(* CoDeSys 2.3.9.41 project: warm.pro *)
(* Libraries: STANDARD.LIB 4.10.05 10:14:46, IECSFC.LIB 13.4.06 14:51:28, SYSLIBTIME.LIB 20.2.06 13:31:16, SYSTASKINFO.LIB 20.2.06 13:31:38, ANALYZATION.LIB 5.10.99 08:05:06, SYSLIBCALLBACK.LIB 20.2.06 13:31:08 *)

(* PLC configuration (modules and I/O channels)
AT %IX0.0 [BitInput]
AT %IX0.1 [BitInput]
AT %IX0.2 [BitInput]
AT %IX0.3 [BitInput]
AT %IX0.4 [BitInput]
AT %IX0.5 [BitInput]
DO0_nurtureValve AT %QX1.0 [BitOutput]
DO1_genatsuValve AT %QX1.1 [BitOutput]
AT %QX1.2 [BitOutput]
AT %QX1.3 [BitOutput]
Special output [ID104] node 2, in %IB2 out %QB2 {Visibility = No; PinCount = 1}
  AT %QX2.0 [BitOutput] Special output
AI0_presIN AT %ID3.0 [FloatInput] Value
AT %IW3.1 [WordInput] Circular time
Analog Input [ID107] node 0, in %IB3.0 out %QB3.0
AI1_presOUT AT %ID4.0 [FloatInput] Value
AT %IW4.1 [WordInput] Circular time
Analog Input [ID107] node 0, in %IB4.0 out %QB4.0
AI2_outsideTemp AT %ID5.0 [FloatInput] Value
AT %IW5.1 [WordInput] Circular time
Analog Input [ID107] node 0, in %IB5.0 out %QB5.0
AT %ID6.0 [FloatInput] Value
AT %IW6.1 [WordInput] Circular time
Analog Input [ID107] node 0, in %IB6.0 out %QB6.0
Analog output [ID106] node 7, in %IB7 out %QB7 {DAC_Type = Voltage 0-10 B; Analog_offset_correction = 0; Analog_full_range_correction = 0; SafeValueFloat = 0; Visibility = No}
  AT %QD7.0 [FloatOutput] Value
Analog output [ID106] node 8, in %IB8 out %QB8 {DAC_Type = Voltage 0-10 B; Analog_offset_correction = 0; Analog_full_range_correction = 0; SafeValueFloat = 0; Visibility = No}
  AT %QD8.0 [FloatOutput] Value
ModBus (Master) [MODBUS_MASTER_ID450] node 9, in %IB9 out %QB9 {Visibility = No}
  AT %QD9.0 [DWordOutput] Last address
  AT %QW9.1 [WordOutput] Last error
  RS-485-1 [COM1_USART] node 0, in %IB9.0 out %QB9.0 {CommunicationSpeed = 11520; Parity = NO PARITY CHECK; BitLength = 8 bits; StopLength = Two stop bits; InterfaceType = RS485; FrameOriented = RTU; Timeout = 0; Visibility = No}
  Universal Modbus device [ID2000] node 1, in %IB9.1 out %QB9.1 {ModuleIP = 10:0:0:223; ServiceTimeout = 150; TCPport = 502; NetMode = Serial; ModuleSlaveAddress = 3; RequestType = By poll time; PeriodOfService = 3000; Visibility = No; RepeatCounter = 0; ByteSequence = Native}
    AT %QB9.1.0 [ComChannel] Command (0xff - Start)
trm1_temperature AT %IW9.1.0.0 [WordInput]
trm1_setpoint AT %IW9.1.1.0 [WordInput]
trm1_state AT %IW9.1.2.0 [WordInput]
trm1_writeSetpoint AT %QW9.1.3.0 [WordOutput]
Universal Modbus device [ID2000] node 2, in %IB9.2 out %QB9.2 {ModuleIP = 10:0:0:223; ServiceTimeout = 150; TCPport = 502; NetMode = Serial; ModuleSlaveAddress = 4; RequestType = By poll time; PeriodOfService = 3000; Visibility = No; RepeatCounter = 0; ByteSequence = Native}
  AT %QB9.2.0 [ComChannel] Command (0xff - Start)
trm2_temperature AT %IW9.2.0.0 [WordInput]
trm2_setpoint AT %IW9.2.1.0 [WordInput]
trm2_state AT %IW9.2.2.0 [WordInput]
trm2_writeSetpoint AT %QW9.2.3.0 [WordOutput]
Universal Modbus device [ID2000] node 3, in %IB9.3 out %QB9.3 {ModuleIP = 10:0:0:223; ServiceTimeout = 150; TCPport = 502; NetMode = Serial; ModuleSlaveAddress = 5; RequestType = By poll time; PeriodOfService = 2000; Visibility = No; RepeatCounter = 0; ByteSequence = Trace_mode}
  AT %QB9.3.0 [ComChannel] Command (0xff - Start)
fc_frequency AT %IW9.3.0.0 [WordInput]
fc_setpoint AT %ID9.3.1.0 [DWordInput]
fc_power AT %ID9.3.2.0 [DWordInput]
fc_currency AT %ID9.3.3.0 [DWordInput]
fc_pressure AT %ID9.3.4.0 [DWordInput]
fc_writeSetpoint AT %QD9.3.5.0 [DWordOutput]
Debug RS-232 [DEBUG_USART] node 0, in %IB10.0.0 out %QB10.0.0 {CommunicationSpeed = 11520; Parity = EVEN; BitLength = 8 bits; StopLength = One stop bit; InterfaceType = RS232; FrameOriented = RTU; Timeout = 0; Visibility = No}
AT %QB10.1.0 [ByteOutput]
AT %QB10.2.0 [ByteOutput]
AT %QB10.3.0 [ByteOutput]
AT %QB10.4.0 [ByteOutput]
pan_weekDays AT %QB10.5.0 [ByteOutput]
pan_holyDays AT %QB10.6.0 [ByteOutput]
2 byte [Register] node 7, in %IB10.7 out %QB10.7
  pan_trm1_temp AT %QW10.7.0 [WordOutput]
  pan_trm1_set AT %QW10.8.0 [WordOutput]
  pan_trm2_temp AT %QW10.9.0 [WordOutput]
  pan_trm2_set AT %QW10.10.0 [WordOutput]
  pan_fc_freq AT %QW10.11.0 [WordOutput]
  pan_fc_curr AT %QW10.12.0 [WordOutput]
  pan_fc_pow AT %QW10.13.0 [WordOutput]
  pan_fc_pres AT %QW10.14.0 [WordOutput]
  pan_fc_set AT %QW10.15.0 [WordOutput]
  pan_presIN_4ma AT %QW10.16.0 [WordOutput]
  pan_presIN_20ma AT %QW10.17.0 [WordOutput]
  pan_presOUT_4ma AT %QW10.18.0 [WordOutput]
  pan_presOUT_20ma AT %QW10.19.0 [WordOutput]
  pan_weekday_set AT %QW10.20.0 [WordOutput]
  pan_holyday_set AT %QW10.21.0 [WordOutput]
  pan_weekday_onHH AT %QW10.22.0 [WordOutput]
  pan_weekday_onMM AT %QW10.23.0 [WordOutput]
  pan_holyday_onHH AT %QW10.24.0 [WordOutput]
  pan_holyday_onMM AT %QW10.25.0 [WordOutput]
  pan_weekday_offHH AT %QW10.26.0 [WordOutput]
  pan_weekday_offMM AT %QW10.27.0 [WordOutput]
  pan_holyday_offHH AT %QW10.28.0 [WordOutput]
  pan_holyday_offMM AT %QW10.29.0 [WordOutput]
  pan_soldierTime AT %QW10.30.0 [WordOutput]
  pan_airLow AT %QW10.31.0 [WordOutput]
  pan_trmLow AT %QW10.32.0 [WordOutput]
  pan_airHigh AT %QW10.33.0 [WordOutput]
  pan_trmHigh AT %QW10.34.0 [WordOutput]
  pan_nurtureHigh AT %QW10.35.0 [WordOutput]
  pan_nurtureLow AT %QW10.36.0 [WordOutput]
  pan_genatsuHigh AT %QW10.37.0 [WordOutput]
  pan_genatsuLow AT %QW10.38.0 [WordOutput]
  pan_presIN AT %QW10.39.0 [WordOutput]
  pan_presOUT AT %QW10.40.0 [WordOutput]
  pan_outsideTemp AT %QW10.41.0 [WordOutput]
  pan_tempShift AT %QW10.42.0 [WordOutput]
  pan_currHH AT %QW10.43.0 [WordOutput]
  pan_currMIN AT %QW10.44.0 [WordOutput]
  pan_currSS AT %QW10.45.0 [WordOutput]
  pan_currDD AT %QW10.46.0 [WordOutput]
  pan_currMM AT %QW10.47.0 [WordOutput]
  pan_currYY AT %QW10.48.0 [WordOutput]
  pan_setHH AT %QW10.49.0 [WordOutput]
  pan_setMIN AT %QW10.50.0 [WordOutput]
  pan_setSS AT %QW10.51.0 [WordOutput]
  pan_setDD AT %QW10.52.0 [WordOutput]
  pan_setMM AT %QW10.53.0 [WordOutput]
  pan_setYY AT %QW10.54.0 [WordOutput]
  pan_genatsuOmakeHigh AT %QW10.55.0 [WordOutput]
  ID4002 byte8IB
8%QB
8%MB
8%Mpan_genatsuOmakeLow AT %QW10.56.0 [WordOutput]
*)

(* Global variable list: Global_Variables *)
VAR_GLOBAL
(* Times *)
	GetTime: CurTimeEx;
	TimeAndDate: SystemTimeDate;
	Sys_Time: SysTime64;
END_VAR

(* POU PLC_PRG, ST *)
PROGRAM PLC_PRG
VAR
	NO_FIRST_PASS : BOOL := FALSE;

	trmGvs_setpoint, trmHeat_setpoint : WORD;
	fc_setpoint : WORD;

	presIN, presIN_4ma, presIN_20ma : WORD;
	presOUT, presOUT_4ma, presOUT_20ma : WORD;

	weekday_setpoint, holyday_setpoint : WORD;
	weekday_byTime, holyday_byTime : BOOL;
	weekday_onHH, holyday_onHH : WORD;
	weekday_onMM, holyday_onMM : WORD;
	weekday_offHH, holyday_offHH : WORD;
	weekday_offMM, holyday_offMM : WORD;

	weekDays, holyDays : WORD;
	newWeekFlag, newHolyFlag : BOOL;

	HeatStart, HeatStarted : BOOL;
	outsideTemp : INT;
	nowHoly : BOOL;
	timeToHeatWeek, timeToHeatHoly : BOOL;

	heatStarting : BOOL;
	soldierTime : WORD;
	soldierTimer : TON;
	soldierOver : BOOL;
	fc_start : BOOL;

	(* heating mode *)
	airLow, trmLow : WORD;
	airHigh, trmHigh : WORD;
	modeSetpoint : WORD;

	realOutsideTemp : REAL;
	realAirLow, realTrmLow : REAL;
	realAirHigh, realTrmHigh : REAL;
	realModeSetpoint : REAL;

	cycleToHeatHoly : SPDAYCYCLE;
	cycleToHeatWeek : SPDAYCYCLE;
	holyCycle, weekCycle : REAL;

	(* nurture *)
	duringNurture : BOOL;
	nurtureHigh, nurtureLow : WORD;
	nurtureOutLack, nurtureOutExceed : BOOL;
	nurtureLackTimer : TON;
	nurtureExceedTimer : TON;
	nurtureRun : BOOL;

	(* genatsu *)
	genatsuChuu : BOOL;
	genatsuHigh, genatsuLow : WORD;
	genatsuInLack, genatsuInExceed : BOOL;
	genatsuLackTimer : TON;
	genatsuExceedTimer : TON;
	genatsuRun : BOOL;

	(* genatsu omake *)
	genatsuOmakeChuu : BOOL;
	genatsuOmakeHigh, genatsuOmakeLow : WORD;
	genatsuOmakeOutLack, genatsuOmakeOutExceed : BOOL;
	genatsuOmakeLackTimer : TON;
	genatsuOmakeExceedTimer : TON;
	genatsuOmakeRun : BOOL;

	(* outside temp *)
	tempShift : INT;

END_VAR
VAR RETAIN
	save_trmGvs_setpoint, save_trmHeat_setpoint : WORD;
	save_fc_setpoint : WORD;

	save_presIN_4ma, save_presIN_20ma : WORD;
	save_presOUT_4ma, save_presOUT_20ma : WORD;

	save_weekday_setpoint, save_holyday_setpoint : WORD;
	save_weekday_byTime, save_holyday_byTime : BOOL;
	save_weekday_onHH, save_holyday_onHH : WORD;
	save_weekday_onMM, save_holyday_onMM : WORD;
	save_weekday_offHH, save_holyday_offHH : WORD;
	save_weekday_offMM, save_holyday_offMM : WORD;

	save_weekDays, save_holyDays : WORD;

	save_soldierTime : WORD;

	save_airLow, save_trmLow : WORD;
	save_airHigh, save_trmHigh : WORD;

	save_nurtureHigh, save_nurtureLow : WORD;
	save_genatsuHigh, save_genatsuLow : WORD;
	save_genatsuOmakeHigh, save_genatsuOmakeLow : WORD;

	save_nurtureRun, save_genatsuRun, save_genatsuOmakeRun : BOOL;

	save_tempShift : WORD;

END_VAR
IF NO_FIRST_PASS = FALSE THEN
			WithdrawRetain;
			NO_FIRST_PASS := TRUE;
END_IF;

Defaults;

SaveNewValue;

Times;

Calibration;

IF nurtureRun THEN
	Nurture;
ELSE
	duringNurture := FALSE;
END_IF;

IF genatsuRun THEN
	Genatsu;
ELSE
	genatsuChuu := FALSE;
END_IF;

TempMode;

Heating;

Transfer;
END_PROGRAM
ACTION Calibration:
presIN := presIN_4ma  + ( REAL_TO_INT( AI0_presIN * 100 ) - 400 ) * ( presIN_20ma - presIN_4ma ) / 1600; (* wordpres := .... точность 0.01 *)

IF AI0_presIN < 4.0 THEN
	presIN := 0;
END_IF;

presOUT := presOUT_4ma  + ( REAL_TO_INT( AI1_presOUT * 100 ) - 400 ) * ( presOUT_20ma - presOUT_4ma ) / 1600; (* wordpres := .... точность 0.01 *)

IF AI1_presOUT < 4.0 THEN
	presOUT := 0;
END_IF;

outsideTemp :=  REAL_TO_INT ( AI2_outsideTemp  * 100 ) + tempShift;
END_ACTION
ACTION Defaults:
IF pan_trm1_set = 0 THEN
	pan_trm1_set := 550;
END_IF;

IF pan_trm2_set = 0 THEN
	pan_trm2_set := 600;
END_IF;

IF pan_fc_set = 0 THEN
	pan_fc_set := 5000;
END_IF;


IF pan_presIN_20ma = 0 THEN
	pan_presIN_20ma := 1975;
END_IF;

IF pan_presOUT_20ma = 0 THEN
	pan_presOUT_20ma := 1785;
END_IF;


IF pan_nurtureHigh = 0 THEN
	pan_nurtureHigh := 270;
END_IF;

IF pan_nurtureLow = 0 THEN
	pan_nurtureLow := 230;
END_IF;

IF pan_genatsuHigh = 0 THEN
	pan_genatsuHigh := 530;
END_IF;

IF pan_genatsuLow = 0 THEN
	pan_genatsuLow := 500;
END_IF;
END_ACTION
ACTION DetermineHoly:
CASE TimeAndDate.DayOfWeek OF
	1 : IF hMON
	     	THEN nowHoly := TRUE;
		ELSE nowHoly := FALSE;
	     END_IF;

	2 : IF hTUE
	     	THEN nowHoly := TRUE;
		ELSE nowHoly := FALSE;
	     END_IF;

      3 : IF hWED
	     	THEN nowHoly := TRUE;
		ELSE nowHoly := FALSE;
	     END_IF;

      4 : IF hTHU
	     	THEN nowHoly := TRUE;
		ELSE nowHoly := FALSE;
	     END_IF;

      5 : IF hFRI
	     	THEN nowHoly := TRUE;
		ELSE nowHoly := FALSE;
	     END_IF;

      6 : IF hSAT
	     	THEN nowHoly := TRUE;
		ELSE nowHoly := FALSE;
	     END_IF;

      0 : IF hSUN
	     	THEN nowHoly := TRUE;
		ELSE nowHoly := FALSE;
	     END_IF;
END_CASE;
END_ACTION
ACTION Genatsu:
IF presIN > genatsuHigh THEN
	genatsuInExceed := TRUE;
ELSE
	genatsuInExceed := FALSE;
END_IF;

IF presIN < genatsuLow THEN
	genatsuInLack := TRUE;
ELSE
	genatsuInLack := FALSE;
END_IF;

genatsuExceedTimer ( IN := genatsuInExceed, PT := T#1s );

IF genatsuExceedTimer.Q OR genatsuChuu THEN
	genatsuChuu := TRUE;
END_IF;

genatsuLackTimer ( IN := genatsuInLack, PT := T#1s );

IF genatsuLackTimer.Q THEN
	genatsuChuu := FALSE;
END_IF;

(* OMAKE *)

IF presOUT > genatsuOmakeHigh THEN
	genatsuOmakeOutExceed := TRUE;
ELSE
	genatsuOmakeOutExceed := FALSE;
END_IF;

IF presOUT < genatsuOmakeLow THEN
	genatsuOmakeOutLack := TRUE;
ELSE
	genatsuOmakeOutLack := FALSE;
END_IF;

genatsuOmakeExceedTimer ( IN := genatsuOmakeOutExceed, PT := T#1s );

IF genatsuOmakeExceedTimer.Q OR genatsuOmakeChuu THEN
	genatsuOmakeChuu := TRUE;
END_IF;

genatsuOmakeLackTimer ( IN := genatsuOmakeOutLack, PT := T#1s );

IF genatsuOmakeLackTimer.Q THEN
	genatsuOmakeChuu := FALSE;
END_IF;
END_ACTION
ACTION Heating:
IF newWeekFlag THEN
	newWeekFlag := FALSE;
	Weekcheck;
END_IF;

IF newHolyFlag THEN
	newHolyFlag := FALSE;
	Holycheck;
END_IF;

(* проверка условий запуска *)

DetermineHoly;


IF nowHoly THEN
	cycleToHeatHoly( firstSetpoint := 1.0, secondSetpoint := 2.0,
						spHHfirst := holyday_onHH, spMMfirst := holyday_onMM,
						spHHsecond := holyday_offHH, spMMsecond := holyday_offMM,
						HH := TimeAndDate.Hour, MM := TimeAndDate.Minute,

						setpoint => holyCycle );

	IF holyCycle = 1.0 THEN
		timeToHeatHoly := TRUE;
	ELSE
		timeToheatHoly := FALSE;
	END_IF;
(*
	IF ( holyday_onHH = TimeAndDate.Hour ) AND ( holyday_onMM = TimeAndDate.Minute ) AND ( TimeAndDate.Second = 0 )
		THEN timeToHeatHoly := TRUE;
	END_IF;

	IF ( holyday_offHH = TimeAndDate.Hour ) AND ( holyday_offMM = TimeAndDate.Minute ) AND ( TimeAndDate.Second = 0 )
		THEN timeToHeatHoly := FALSE;
	END_IF;
*)
ELSE
	cycleToHeatWeek( firstSetpoint := 1.0, secondSetpoint := 2.0,
						spHHfirst := weekday_onHH, spMMfirst := weekday_onMM,
						spHHsecond := weekday_offHH, spMMsecond := weekday_offMM,
						HH := TimeAndDate.Hour, MM := TimeAndDate.Minute,

						setpoint => weekCycle );

	IF weekCycle = 1.0 THEN
		timeToHeatWeek := TRUE;
	ELSE
		timeToheatWeek := FALSE;
	END_IF;
(*
	IF ( weekday_onHH = TimeAndDate.Hour ) AND ( weekday_onMM = TimeAndDate.Minute ) AND ( TimeAndDate.Second = 0 )
		THEN timeToHeatWeek := TRUE;
	END_IF;

	IF ( weekday_offHH = TimeAndDate.Hour ) AND ( weekday_offMM = TimeAndDate.Minute ) AND ( TimeAndDate.Second = 0 )
		THEN timeToHeatWeek := FALSE;
	END_IF;
*)
END_IF;


IF nowHoly THEN
	IF holyday_byTime THEN
		IF ( outsideTemp < holyday_setpoint ) AND  timeToHeatHoly THEN
			HeatStart := TRUE;
		ELSE
			HeatStart := FALSE;
		END_IF;
	ELSE
		IF outsideTemp < holyday_setpoint THEN
			HeatStart := TRUE;
		ELSE
			HeatStart := FALSE;
		END_IF;
	END_IF;
ELSE
	IF weekday_byTime THEN
		IF ( outsideTemp < weekday_setpoint ) AND  timeToHeatWeek THEN
			HeatStart := TRUE;
		ELSE
			HeatStart := FALSE;
		END_IF;
	ELSE
		IF outsideTemp < weekday_setpoint THEN
			HeatStart := TRUE;
		ELSE
			HeatStart := FALSE;
		END_IF;
	END_IF;
END_IF;


(* пуск системы отопления *)
(* разобраться с типами soldierTimer(IN:= HeatStart, PT:=soldierTime, Q=>soldierOver, ET=> ); *)

IF HeatStart AND NOT HeatStarted THEN
	fc_start := TRUE;
	heatStarting := TRUE;
	IF soldierOver THEN
		heatStarting := FALSE;
		HeatStarted := TRUE;
	END_IF;
END_IF;

(* останов системы отопления *)
IF NOT HeatStart AND HeatStarted THEN
	fc_start := FALSE;

END_IF;

IF heatStarting THEN
	trm1_writeSetpoint := 1000;
ELSE
	trm1_writeSetpoint := trmGvs_setpoint;
END_IF;
END_ACTION
ACTION Holycheck:
IF wMON = hMON THEN
	wMON := NOT hMON;
END_IF;

IF wTUE = hTUE THEN
	wTUE := NOT hTUE;
END_IF;

IF wWED = hWED THEN
	wWED := NOT hWED;
END_IF;

IF wTHU = hTHU THEN
	wTHU := NOT hTHU;
END_IF;

IF wFRI = hFRI THEN
	wFRI := NOT hFRI;
END_IF;

IF wSAT = hSAT THEN
	wSAT := NOT hSAT;
END_IF;

IF wSUN = hSUN THEN
	hSUN := NOT wSUN;
END_IF;
END_ACTION
ACTION Input:
;
END_ACTION
ACTION Nurture:
IF presOUT < nurtureLow THEN
	nurtureOutLack := TRUE;
ELSE
	nurtureOutLack := FALSE;
END_IF;

IF presOUT > nurtureHigh THEN
	nurtureOutExceed := TRUE;
ELSE
	nurtureOutExceed := FALSE;
END_IF;

nurtureLackTimer ( IN := nurtureOutLack, PT := T#1s );

IF nurtureLackTimer.Q OR duringNurture THEN
	duringNurture := TRUE;
END_IF;

nurtureExceedTimer ( IN := nurtureOutExceed, PT := T#1s );

IF nurtureExceedTimer.Q THEN
	duringNurture := FALSE;
END_IF;
END_ACTION
ACTION SaveNewValue:
IF pan_trm1_set <> trmGvs_setpoint THEN
	save_trmGvs_setpoint := pan_trm1_set;
	trmGvs_setpoint := pan_trm1_set;
END_IF;

IF pan_trm2_set <> trmHeat_setpoint THEN
	save_trmHeat_setpoint := pan_trm2_set;
	trmHeat_setpoint := pan_trm2_set;
END_IF;

IF pan_fc_set <> fc_setpoint THEN
	save_fc_setpoint := pan_fc_set;
	fc_setpoint := pan_fc_set;
END_IF;

IF pan_presIN_4ma <> presIN_4ma THEN
	save_presIN_4ma := pan_presIN_4ma;
	presIN_4ma := pan_presIN_4ma;
END_IF;

IF pan_presIN_20ma <> presIN_20ma THEN
	save_presIN_20ma := pan_presIN_20ma;
	presIN_20ma := pan_presIN_20ma;
END_IF;

IF pan_presOUT_4ma <> presOUT_4ma THEN
	save_presOUT_4ma := pan_presOUT_4ma;
	presOUT_4ma := pan_presOUT_4ma;
END_IF;

IF pan_presOUT_20ma <> presOUT_20ma THEN
	save_presOUT_20ma := pan_presOUT_20ma;
	presOUT_20ma := pan_presOUT_20ma;
END_IF;

IF pan_weekday_set <> weekday_setpoint THEN
	save_weekday_setpoint := pan_weekday_set;
	weekday_setpoint := pan_weekday_set;
END_IF;

IF pan_holyday_set <> holyday_setpoint THEN
	save_holyday_setpoint := pan_holyday_set;
	holyday_setpoint := pan_holyday_set;
END_IF;

IF pan_weekday_byTime <> weekday_byTime THEN
	save_weekday_byTime := pan_weekday_byTime;
	weekday_byTime := pan_weekday_byTime;
END_IF;

IF pan_holyday_byTime <> holyday_byTime THEN
	save_holyday_byTime := pan_holyday_byTime;
	holyday_byTime := pan_holyday_byTime;
END_IF;

IF pan_weekday_onHH <> weekday_onHH THEN
	save_weekday_onHH := pan_weekday_onHH;
	weekday_onHH := pan_weekday_onHH;
END_IF;

IF pan_weekday_onMM <> weekday_onMM THEN
	save_weekday_onMM := pan_weekday_onMM;
	weekday_onMM := pan_weekday_onMM;
END_IF;

IF pan_holyday_onHH <> holyday_onHH THEN
	save_holyday_onHH := pan_holyday_onHH;
	holyday_onHH := pan_holyday_onHH;
END_IF;

IF pan_holyday_onMM <> holyday_onMM THEN
	save_holyday_onMM := pan_holyday_onMM;
	holyday_onMM := pan_holyday_onMM;
END_IF;


IF pan_weekday_offHH <> weekday_offHH THEN
	save_weekday_offHH := pan_weekday_offHH;
	weekday_offHH := pan_weekday_offHH;
END_IF;

IF pan_weekday_offMM <> weekday_offMM THEN
	save_weekday_offMM := pan_weekday_offMM;
	weekday_offMM := pan_weekday_offMM;
END_IF;

IF pan_holyday_offHH <> holyday_offHH THEN
	save_holyday_offHH := pan_holyday_offHH;
	holyday_offHH := pan_holyday_offHH;
END_IF;

IF pan_holyday_offMM <> holyday_offMM THEN
	save_holyday_offMM := pan_holyday_offMM;
	holyday_offMM := pan_holyday_offMM;
END_IF;

IF BYTE_TO_WORD ( pan_weekDays ) <> weekDays THEN
	save_weekDays := BYTE_TO_WORD ( pan_weekDays );
	weekDays := BYTE_TO_WORD ( pan_weekDays );
	newWeekFlag := TRUE;
END_IF;

IF BYTE_TO_WORD ( pan_holyDays ) <> holyDays THEN
	save_holyDays := BYTE_TO_WORD ( pan_holyDays );
	holyDays := BYTE_TO_WORD ( pan_holyDays );
	newHolyFlag := TRUE;
END_IF;

IF pan_soldierTime <> soldierTime THEN
	save_soldierTime := pan_soldierTime;
	soldierTime := pan_soldierTime;
END_IF;

IF pan_airLow <> airLow THEN
	save_airLow := pan_airLow;
	airLow := pan_airLow;
END_IF;

IF pan_trmLow <> trmLow THEN
	save_trmLow := pan_trmLow;
	trmLow := pan_trmLow;
END_IF;

IF pan_airHigh <> airHigh THEN
	save_airHigh := pan_airHigh;
	airHigh := pan_airHigh;
END_IF;

IF pan_trmHigh <> trmHigh THEN
	save_trmHigh := pan_trmHigh;
	trmHigh := pan_trmHigh;
END_IF;

IF pan_nurtureHigh <> nurtureHigh THEN
	save_nurtureHigh := pan_nurtureHigh;
	nurtureHigh := pan_nurtureHigh;
END_IF;

IF pan_nurtureLow <> nurtureLow THEN
	save_nurtureLow := pan_nurtureLow;
	nurtureLow := pan_nurtureLow;
END_IF;

IF pan_genatsuHigh <> genatsuHigh THEN
	save_genatsuHigh := pan_genatsuHigh;
	genatsuHigh := pan_genatsuHigh;
END_IF;

IF pan_genatsuLow <> genatsuLow THEN
	save_genatsuLow := pan_genatsuLow;
	genatsuLow := pan_genatsuLow;
END_IF;

IF pan_genatsuOmakeHigh <> genatsuOmakeHigh THEN
	save_genatsuOmakeHigh := pan_genatsuOmakeHigh;
	genatsuOmakeHigh := pan_genatsuOmakeHigh;
END_IF;

IF pan_genatsuOmakeLow <> genatsuOmakeLow THEN
	save_genatsuOmakeLow := pan_genatsuOmakeLow;
	genatsuOmakeLow := pan_genatsuOmakeLow;
END_IF;

IF pan_nurtureRun THEN
	save_nurtureRun := TRUE;
	nurtureRun := TRUE;
ELSE
	save_nurtureRun := FALSE;
	nurtureRun := FALSE;
END_IF;

IF pan_genatsuRun THEN
	save_genatsuRun := TRUE;
	genatsuRun := TRUE;
ELSE
	save_genatsuRun := FALSE;
	genatsuRun := FALSE;
END_IF;

IF pan_genatsuOmakeRun THEN
	save_genatsuOmakeRun := TRUE;
	genatsuOmakeRun := TRUE;
ELSE
	save_genatsuOmakeRun := FALSE;
	genatsuOmakeRun := FALSE;
END_IF;

IF WORD_TO_INT ( pan_tempShift ) <> tempShift THEN
	save_tempShift := pan_tempShift;
	tempShift := WORD_TO_INT ( pan_tempShift );
END_IF;
END_ACTION
ACTION TempMode:
(* realOutsideTemp *)
realAirLow :=   WORD_TO_REAL ( airLow ) / 100;
realTrmLow := WORD_TO_REAL ( trmLow ) / 100;
realAirHigh :=   WORD_TO_REAL ( airHigh )  / 100;
realTrmHigh := WORD_TO_REAL ( trmHigh ) / 100;

realModeSetpoint := ( ( realOutsideTemp * ( realTrmHigh - realTrmLow ) ) - ( realTrmHigh * realAirLow ) + ( realTrmLow * realAirHigh ) ) / ( realAirHigh - realAirLow );

modeSetpoint := REAL_TO_WORD ( realModeSetpoint * 100 );
END_ACTION
ACTION Times:
TimeAndDate.Day :=0;
TimeAndDate.DayOfWeek :=0;
TimeAndDate.dwHighMsec :=0;
TimeAndDate.dwLowMSecs :=0;
TimeAndDate.Milliseconds :=0;
TimeAndDate.Minute :=0;
TimeAndDate.Second :=0;
TimeAndDate.Hour :=0;
TimeAndDate.Year :=0;
TimeAndDate.Month :=0;
Sys_time.ulHigh :=0;
Sys_time.ulLow :=0;
GetTime (SystemTime:=Sys_Time , TimeDate:= TimeAndDate);


IF pan_setTime THEN
	TimeAndDate.Minute:=pan_setMIN;
	TimeAndDate.Second:=pan_setSS;
	TimeAndDate.Hour:=pan_setHH;
	TimeAndDate.Day:=pan_setDD;
	TimeAndDate.Month:=pan_setMM;
	TimeAndDate.Year:=pan_setYY;
	GetTime (SystemTime:=Sys_Time , TimeDate:= TimeAndDate);

	pan_setTime := FALSE;
END_IF;
END_ACTION
ACTION Transfer:
pan_presIN := presIN;
pan_presOUT := presOUT;

IF duringNurture THEN
	DO0_nurtureValve := TRUE;
	pan_nurtureValve := TRUE;
ELSE
	DO0_nurtureValve := FALSE;
	pan_nurtureValve := FALSE;
END_IF;

IF genatsuChuu OR genatsuOmakeChuu THEN
	DO1_genatsuValve := TRUE;
	pan_genatsuValve := TRUE;
ELSE
	DO1_genatsuValve := FALSE;
	pan_genatsuValve := FALSE;
END_IF;

(* DANFOSS *)
pan_fc_freq :=  fc_frequency;
pan_fc_curr := DWORD_TO_WORD ( fc_currency );
pan_fc_pow := DWORD_TO_WORD ( fc_power );
pan_fc_pres := DWORD_TO_WORD ( fc_pressure );

fc_writeSetpoint := WORD_TO_DWORD ( pan_fc_set );

(* TRM *)
pan_trm1_temp := trm1_temperature;
pan_trm2_temp := trm2_temperature;

trm1_writeSetpoint :=  pan_trm1_set;
trm2_writeSetpoint := pan_trm2_set;

IF trm1_state = 1000 THEN
	pan_trm1_state := TRUE;
	pan_trm1_valve := FALSE;
ELSE
	pan_trm1_state := FALSE;
	pan_trm1_valve := TRUE;
END_IF;

IF trm2_state = 1000 THEN
	pan_trm2_state := TRUE;
	pan_trm2_valve := FALSE;
ELSE
	pan_trm2_state := FALSE;
	pan_trm2_valve := TRUE;
END_IF;

(* outside temp *)
pan_outsideTemp := INT_TO_WORD ( outsideTemp );
END_ACTION
ACTION Weekcheck:
IF wMON = hMON THEN
	hMON := NOT wMON;
END_IF;

IF wTUE = hTUE THEN
	hTUE := NOT wTUE;
END_IF;

IF wWED = hWED THEN
	hWED := NOT wWED;
END_IF;

IF wTHU = hTHU THEN
	hTHU := NOT wTHU;
END_IF;

IF wFRI = hFRI THEN
	hFRI := NOT wFRI;
END_IF;

IF wSAT = hSAT THEN
	hSAT := NOT wSAT;
END_IF;

IF wSUN = hSUN THEN
	hSUN := NOT wSUN;
END_IF;
END_ACTION
ACTION WithdrawRetain:
trmGvs_setpoint := save_trmGvs_setpoint;
trmHeat_setpoint := save_trmHeat_setpoint;
pan_trm1_set := save_trmGvs_setpoint;
pan_trm2_set := save_trmHeat_setpoint;
fc_setpoint := save_fc_setpoint;
pan_fc_set := save_fc_setpoint;

presIN_4ma := save_presIN_4ma;
presIN_20ma := save_presIN_20ma;
presOUT_4ma := save_presOUT_4ma;
presOUT_20ma := save_presOUT_20ma;

pan_presIN_4ma := save_presIN_4ma;
pan_presIN_20ma := save_presIN_20ma;
pan_presOUT_4ma := save_presOUT_4ma;
pan_presOUT_20ma := save_presOUT_20ma;


weekday_setpoint :=  save_weekday_setpoint;
holyday_setpoint :=   save_holyday_setpoint;
weekday_byTime := save_weekday_byTime;
holyday_byTime :=  save_holyday_byTime;
weekday_onHH := save_weekday_onHH;
holyday_onHH :=  save_holyday_onHH;
weekday_onMM := save_weekday_onMM;
holyday_onMM :=   save_holyday_onMM;
weekday_offHH := save_weekday_offHH;
holyday_offHH :=   save_holyday_offHH;
weekday_offMM := save_weekday_offMM;
holyday_offMM :=   save_holyday_offMM;

weekDays := save_weekDays;
holyDays :=  save_holyDays;

soldierTime := save_soldierTime;

airLow := save_airLow;
trmLow := save_trmLow;
airHigh := save_airHigh;
trmHigh := save_trmHigh;

nurtureHigh := save_nurtureHigh;
nurtureLow := save_nurtureLow;
genatsuHigh := save_genatsuHigh;
genatsuLow := save_genatsuLow;

pan_nurtureHigh := save_nurtureHigh;
pan_nurtureLow := save_nurtureLow;
pan_genatsuHigh := save_genatsuHigh;
pan_genatsuLow := save_genatsuLow;


pan_genatsuOmakeHigh := save_genatsuOmakeHigh;
pan_genatsuOmakeLow := save_genatsuOmakeLow;

pan_nurtureRun := FALSE;
pan_genatsuRun := FALSE;
pan_genatsuOmakeRun := FALSE;
(*
IF save_nurtureRun THEN
	pan_nurtureRun := TRUE;
ELSE
	pan_nurtureRun := FALSE;
END_IF;

IF save_genatsuRun THEN
	pan_genatsuRun := TRUE;
ELSE
	pan_genatsuRun := FALSE;
END_IF;
*)
pan_tempShift := save_tempShift;
END_ACTION

(* POU SPDAYCYCLE, ST *)
FUNCTION_BLOCK SPDAYCYCLE
VAR_INPUT
	firstSetpoint : REAL;
	secondSetpoint : REAL;
	spHHfirst : WORD;
	spMMfirst : WORD;
	spHHsecond : WORD;
	spMMsecond : WORD;
	HH, MM : WORD;
END_VAR
VAR_OUTPUT
	setpoint : REAL;
END_VAR
VAR
END_VAR
IF spHHsecond > spHHfirst THEN
	IF HH = spHHsecond AND MM >= spMMsecond THEN
		setpoint := secondSetpoint;
	END_IF;
	IF HH > spHHsecond AND HH > spHHfirst THEN
		setpoint := secondSetpoint;
	END_IF;
	IF HH >= 0 AND HH < spHHfirst THEN
		setpoint := secondSetpoint;
	END_IF;
	IF HH = spHHfirst AND MM < spMMfirst THEN
		setpoint := secondSetpoint;
	END_IF;
	IF HH = spHHfirst AND MM >= spMMfirst THEN
		setpoint := firstSetpoint;
	END_IF;
	IF HH > spHHfirst AND HH < spHHsecond THEN
		setpoint := firstSetpoint;
	END_IF;
	IF HH = spHHsecond AND MM < spMMsecond THEN
		setpoint := firstSetpoint;
	END_IF;
END_IF;

IF spHHsecond < spHHfirst THEN
	IF HH = spHHsecond AND MM >= spMMsecond THEN
		setpoint := secondSetpoint;
	END_IF;
	IF HH > spHHsecond AND HH < spHHfirst THEN
		setpoint := secondSetpoint;
	END_IF;
	IF HH = spHHfirst AND MM < spMMfirst THEN
		setpoint := secondSetpoint;
	END_IF;
	IF HH = spHHfirst AND MM >= spMMfirst THEN
		setpoint := firstSetpoint;
	END_IF;
	IF HH > spHHfirst THEN
		setpoint := firstSetpoint;
	END_IF;
	IF HH >= 0 AND spHHsecond > 0 THEN
		setpoint := firstSetpoint;
	END_IF;
	IF HH = spHHsecond AND MM < spMMsecond THEN
		setpoint := firstSetpoint;
	END_IF;
END_IF;
END_FUNCTION_BLOCK

(* POU CALIBRATION, ST *)
FUNCTION_BLOCK CALIBRATION
VAR_INPUT
	AI_RAW : REAL;
	w2d_sensorBottom : WORD;
	w2d_sensorTop : WORD;
	r_sensorBottom : REAL;
	r_sensorTop : REAL;

	w2d_scaleBottom : WORD;
	w2d_scaleTop : WORD;
	r_scaleBottom : REAL;
	r_scaleTop : REAL;
END_VAR
VAR_OUTPUT
	r_scaled : REAL;
	w2d_scaled : WORD;
END_VAR
VAR
END_VAR
(* Result = n2 + ( Input - n1 ) * ( ( m2 - n2 ) / ( m1 - n1 ) ) *)

w2d_scaled := w2d_scaleBottom  + ( REAL_TO_INT( AI_RAW * 100 ) - w2d_sensorBottom ) * ( ( w2d_scaleTop - w2d_scaleBottom ) / ( w2d_sensorTop - w2d_sensorBottom ) );

r_scaled := r_scaleBottom  + ( AI_RAW - r_sensorBottom ) * ( ( r_scaleTop - r_scaleBottom ) / ( r_sensorTop - r_sensorBottom ) );
END_FUNCTION_BLOCK
